// TIA Portal project "FactoryIO_Template_S7-1200_V16_V16" (V16)
// Vorlageprojekt für das Buch mit Zielsystem S7-1200

(* hardware
DEVICE "S7-1200-Station_1"  S7-1200 Station
   slot 0: "Baugruppenträger_0"  Rack  V1.0
   slot 1: "PLC_1"  CPU 1211C DC/DC/DC  6ES7 211-1AE40-0XB0  V4.1
*)

// ===== PLC "PLC_1"  CPU 1211C DC/DC/DC =====

VAR_GLOBAL   // PLC tag table "Standard-Variablentabelle"
   "Belt (6m) 1" AT %A0.0 : Bool;
   "start" AT %E0.0 : Bool;
   "stop" AT %E0.1 : Bool;
   "Tag_4" AT %I10.0 : Bool;
   "Tag_5" AT %Q10.0 : Bool;
   "Tag_6" AT %I10.1 : Bool;
   "X" AT %M0.0 : Bool;
   "vision1(Green)" AT %I0.2 : Bool;
   "belt(2m) 1" AT %Q0.1 : Bool;
   "pusherBack" AT %I0.4 : Bool;
   "pusher1" AT %Q0.5 : Bool;
   "pusher1 F" AT %I0.6 : Bool;
   "vision2(Blue)" AT %I0.3 : Bool;
   "pusher2" AT %Q0.6 : Bool;
   "pusher2 F" AT %I0.7 : Bool;
   "belt(2m)2" AT %Q0.2 : Bool;
   "CCW" AT %Q0.4 : Bool;
   "belt (2m) 3" AT %Q0.3 : Bool;
   "Stop Indicator" AT %Q1.0 : Bool;
   "Start Indicator" AT %Q0.7 : Bool;
END_VAR

FUNCTION "MHJ-PLC-Lab-Function-S71200" : Void   // FC9000, SCL
{ S7_Optimized_Access := 'TRUE' }
VERSION : 0.1
   VAR_TEMP
      rdTimeReturn : Int;
      outputTime : DTL;
      SyncVal : Byte;
      forVal : Int;
      forVal_2 : Int;
      Value : Byte;
   END_VAR
   VAR CONSTANT
      CompVal : Byte := 16#34;
      Value_01 : Byte := 16#11;
      Value_01_DW : DWord := 16#A165_D992;
      Value_02_DW : DWord := 16#58BE_4401;
   END_VAR
BEGIN

   #Value:=PEEK(area := 16#82,
        dbNumber := 0,
        byteOffset := 511);
   #Value := #Value + 1;

   POKE(area := 16#82,
        dbNumber := 0,
        byteOffset := 511,
        value := #Value);

   POKE(area:=16#81,
        dbNumber:=0,
        byteOffset:=1016,
        value:=#Value_01_DW);
   POKE(area := 16#81,
        dbNumber := 0,
        byteOffset := 1020,
        value := #Value_02_DW);

   POKE(area := 16#81,
        dbNumber := 0,
        byteOffset := 511,
        value := B#16#00);

   FOR #forVal := 0 TO 120 DO
       FOR #forVal_2:=0 TO 10 DO
           #rdTimeReturn:=RD_SYS_T(#outputTime);
           #rdTimeReturn := WR_SYS_T(#outputTime);
           #rdTimeReturn := RD_SYS_T(#outputTime);
           #rdTimeReturn := WR_SYS_T(#outputTime);
       END_FOR;
       #SyncVal:= PEEK(area := 16#81,
                      dbNumber := 0,
                      byteOffset := 511);
       IF #SyncVal = #CompVal THEN
          GOTO M_1;
       END_IF;
   END_FOR;
   RETURN;

   M_1:
   POKE(area := 16#81,
        dbNumber := 0,
        byteOffset := 511,
        value := B#16#0);
END_FUNCTION

ORGANIZATION_BLOCK "Main"   // OB1, LAD, ProgramCycle
TITLE = "Main Program Sweep (Cycle)"
{ S7_Optimized_Access := 'TRUE' }
VERSION : 0.1
   VAR_INPUT
      Initial_Call : Bool;   // Initial call of this OB
      Remanence : Bool;   // =True, if remanent data are available
   END_VAR
BEGIN

REGION Network 1: Konnektierungsbaustein für PLC-Lab
   // Im Netzwerk 1 wird der Konnektierungsbaustein für PLC-Lab aufgerufen.
   // Dieser Aufruf darf nicht entfernt werden!
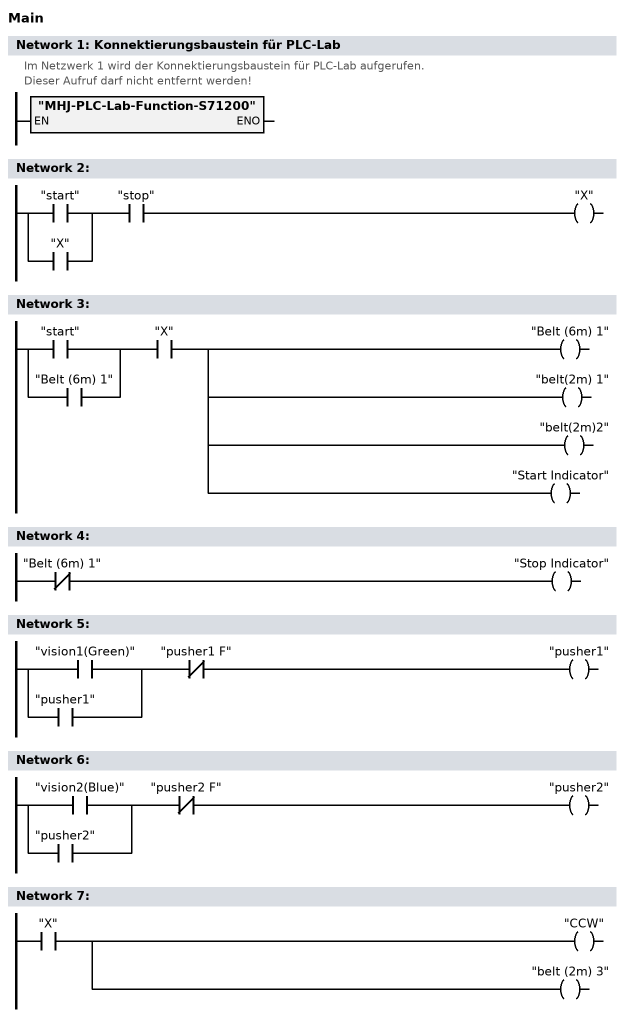
   RUNG wire#powerrail
      "MHJ-PLC-Lab-Function-S71200"()
   END_RUNG
   // the same network as SCL:
   "MHJ-PLC-Lab-Function-S71200"();
END_REGION

REGION Network 2
   RUNG wire#powerrail
      Contact( "start" )
      wire#w1
      Contact( "stop" )
      Coil( "X" )
   END_RUNG
   RUNG wire#powerrail
      Contact( "X" )
   END_RUNG wire#w1
   // the same network as SCL:
   "X" := ("start" OR "X") AND "stop";
END_REGION

REGION Network 3
   RUNG wire#powerrail
      Contact( "start" )
      wire#w1
      Contact( "X" )
      wire#w2
      Coil( "Belt (6m) 1" )
   END_RUNG
   RUNG wire#powerrail
      Contact( "Belt (6m) 1" )
   END_RUNG wire#w1
   RUNG wire#w2
      Coil( "belt(2m) 1" )
   END_RUNG
   RUNG wire#w2
      Coil( "belt(2m)2" )
   END_RUNG
   RUNG wire#w2
      Coil( "Start Indicator" )
   END_RUNG
   // the same network as SCL:
   "Belt (6m) 1" := ("start" OR "Belt (6m) 1") AND "X";
   "belt(2m) 1" := "Belt (6m) 1";
   "belt(2m)2" := "Belt (6m) 1";
   "Start Indicator" := "Belt (6m) 1";
END_REGION

REGION Network 4
   RUNG wire#powerrail
      I_Contact( "Belt (6m) 1" )
      Coil( "Stop Indicator" )
   END_RUNG
   // the same network as SCL:
   "Stop Indicator" := NOT "Belt (6m) 1";
END_REGION

REGION Network 5
   RUNG wire#powerrail
      Contact( "vision1(Green)" )
      wire#w1
      I_Contact( "pusher1 F" )
      Coil( "pusher1" )
   END_RUNG
   RUNG wire#powerrail
      Contact( "pusher1" )
   END_RUNG wire#w1
   // the same network as SCL:
   "pusher1" := ("vision1(Green)" OR "pusher1") AND NOT "pusher1 F";
END_REGION

REGION Network 6
   RUNG wire#powerrail
      Contact( "vision2(Blue)" )
      wire#w1
      I_Contact( "pusher2 F" )
      Coil( "pusher2" )
   END_RUNG
   RUNG wire#powerrail
      Contact( "pusher2" )
   END_RUNG wire#w1
   // the same network as SCL:
   "pusher2" := ("vision2(Blue)" OR "pusher2") AND NOT "pusher2 F";
END_REGION

REGION Network 7
   RUNG wire#powerrail
      Contact( "X" )
      wire#w1
      Coil( "CCW" )
   END_RUNG
   RUNG wire#w1
      Coil( "belt (2m) 3" )
   END_RUNG
   // the same network as SCL:
   "CCW" := "X";
   "belt (2m) 3" := "X";
END_REGION
END_ORGANIZATION_BLOCK